(* IEC 61131-3 sources: teller/JD_Teller_LC2_V11/Class/TanabeCounterSerial, 1 file *)

(* ---- TanabeCounterSerial.st ---- *)
(*!
<Class
	Name               = "TanabeCounterSerial"
	Revision           = "1.0"
	RealtimeTask       = "false"
	CyclicTask         = "true"
	DefCyclictime      = "1 ms"
	BackgroundTask     = "false"
	Sigmatek           = "false"
	OSInterface        = "false"
	HighPriority       = "false"
	Automatic          = "false"
	UpdateMode         = "Prescan"
	SharedCommandTable = "true"
	Objectsize         = "(872,120)">
	<Channels>
		<Server Name="ClassSvr" Visualized="false" Initialize="false" WriteProtected="true" Retentive="false"/>
		<Server Name="iActualProduction" Visualized="false" Initialize="false" WriteProtected="false" Retentive="false"/>
		<Server Name="iBalanceOfProduction" Visualized="false" Initialize="false" WriteProtected="false" Retentive="false"/>
		<Server Name="iConveyorSpeed" Visualized="false" Initialize="false" WriteProtected="false" Retentive="false"/>
		<Server Name="iPlannedProduction" Visualized="false" Initialize="false" WriteProtected="false" Retentive="false"/>
		<Server Name="iProductionSpeed" Visualized="false" Initialize="false" WriteProtected="false" Retentive="false"/>
		<Server Name="sAangepasteWaarde" Visualized="false" Initialize="false" WriteProtected="false" Retentive="false"/>
		<Server Name="sBatch" Visualized="false" Initialize="false" WriteProtected="false" Retentive="false"/>
		<Server Name="sBattingDistance" Visualized="false" Initialize="false" WriteProtected="false" Retentive="false"/>
		<Server Name="sBattingStart" Visualized="false" Initialize="false" WriteProtected="false" Retentive="false"/>
		<Server Name="sBoxLength" Visualized="false" Initialize="false" WriteProtected="false" Retentive="false"/>
		<Server Name="sChangeOfActualQuantity" Visualized="false" Initialize="false" WriteProtected="true" Retentive="false"/>
		<Server Name="sCheckWrittenData" Visualized="false" Initialize="false" WriteProtected="true" Retentive="false"/>
		<Server Name="sClearProdData" Visualized="false" Initialize="false" WriteProtected="true" Retentive="false"/>
		<Server Name="sDateInput" Visualized="false" Initialize="false" WriteProtected="false" Retentive="false"/>
		<Server Name="sLotNo" Visualized="false" Initialize="false" WriteProtected="false" Retentive="false"/>
		<Server Name="sOperatorName" Visualized="false" Initialize="false" WriteProtected="false" Retentive="false"/>
		<Server Name="sProductionQuantity" Visualized="false" Initialize="false" WriteProtected="false" Retentive="false"/>
		<Server Name="sReadAConditionInProgress" Visualized="false" Initialize="false" WriteProtected="true" Retentive="false"/>
		<Server Name="sReturnNak" Visualized="false" Initialize="false" WriteProtected="true" Retentive="false"/>
		<Server Name="sStartingDistanceToConveyor" Visualized="false" Initialize="false" WriteProtected="false" Retentive="false"/>
		<Server Name="sTimeInput" Visualized="false" Initialize="false" WriteProtected="false" Retentive="false"/>
		<Server Name="sWriteProductionData" Visualized="false" Initialize="false" WriteProtected="true" Retentive="false"/>
		<Server Name="verklikker" Visualized="false" Initialize="false" WriteProtected="true" Retentive="false"/>
		<Server Name="Verzenden" Visualized="false" Initialize="false" WriteProtected="false" Retentive="false"/>
		<Client Name="cBatch1" Required="true" Internal="false"/>
		<Client Name="cBatch2" Required="true" Internal="false"/>
		<Client Name="cBattingDistance" Required="true" Internal="false"/>
		<Client Name="cBattingStart" Required="true" Internal="false"/>
		<Client Name="cBoxLength" Required="true" Internal="false"/>
		<Client Name="cCountedBoxes" Required="true" Internal="false"/>
		<Client Name="cPlannedProduction" Required="true" Internal="false"/>
		<Client Name="cStartingDistanceToConveyorRun" Required="true" Internal="false"/>
		<Client Name="FileBase" Required="true" Internal="false"/>
		<Client Name="GetInfo" Required="true" Internal="false"/>
		<Client Name="RxTx" Required="true" Internal="false"/>
		<Client Name="String" Required="true" Internal="false"/>
	</Channels>
	<RevDoku>
		<Owner Company="JD" Author="SV"/>
		<Dokumentation Revision="1" Date="2014-10-13" Author="SV" Company="JD" Description="Class om serieel (RS232) te communiceren met de hoofdcomputer van Tanabe."/>
	</RevDoku>
</Class>
*)
TanabeCounterSerial : CLASS
	TYPE
#pragma pack(push, 1)
	  TypeW : STRUCT  //! <Type Public="true" Name="TypeW"/>
	    Header : ARRAY [0..3] OF CHAR;
	    DateInput : ARRAY [0..6] OF CHAR;
	    TimeInPut : ARRAY [0..6] OF CHAR;
	    ProductionQuantity : ARRAY [0..6] OF CHAR;
	    BoxLength : ARRAY [0..4] OF CHAR;
	    BattingStart : ARRAY [0..3] OF CHAR;
	    BattingDistance : ARRAY [0..3] OF CHAR;
	    Batch : ARRAY [0..2] OF CHAR;
	    LotNo : ARRAY [0..17] OF CHAR;
	    OperatorName : ARRAY [0..8] OF CHAR;
	    StartingDistanceConveyor : ARRAY [0..4] OF CHAR;
	    AlterationOfActualProduction : ARRAY [0..6] OF CHAR;
	    Terminator : CHAR;
	  END_STRUCT;
#pragma pack(pop)
	END_TYPE
  //Servers:
	ClassSvr 	: SvrChCmd_DINT;
	verklikker 	: SvrCh_DINT;
	sReadAConditionInProgress 	: SvrCh_UDINT;
	sWriteProductionData 	: SvrCh_UDINT;
	sCheckWrittenData 	: SvrCh_UDINT;
	sClearProdData 	: SvrCh_UDINT;
	sChangeOfActualQuantity 	: SvrCh_UDINT;
	sReturnNak 	: SvrCh_UDINT;
	iPlannedProduction 	: SvrCh_DINT;
	iBalanceOfProduction 	: SvrCh_DINT;
	iActualProduction 	: SvrCh_DINT;
	iProductionSpeed 	: SvrCh_DINT;
	iConveyorSpeed 	: SvrCh_DINT;
	sDateInput 	: SvrCh_DINT;
	sTimeInput 	: SvrCh_DINT;
	sProductionQuantity 	: SvrCh_DINT;
	sBoxLength 	: SvrCh_DINT;
	sBattingStart 	: SvrCh_DINT;
	sBattingDistance 	: SvrCh_DINT;
	sBatch 	: SvrCh_DINT;
	sLotNo 	: SvrCh_DINT;
	sOperatorName 	: SvrCh_DINT;
	sStartingDistanceToConveyor 	: SvrCh_DINT;
	sAangepasteWaarde 	: SvrCh_DINT;
	Verzenden 	: SvrCh_DINT;
  //Clients:
	GetInfo 	: CltChCmd_TellerClass_Teller;
	RxTx 	: CltChCmd__SerLib;
	String 	: CltChCmd_String;
	FileBase 	: CltChCmd_FileBase;
	cPlannedProduction 	: CltCh_DINT;
	cBoxLength 	: CltCh_DINT;
	cBattingStart 	: CltCh_DINT;
	cBattingDistance 	: CltCh_DINT;
	cBatch1 	: CltCh_DINT;
	cBatch2 	: CltCh_DINT;
	cStartingDistanceToConveyorRun 	: CltCh_DINT;
	cCountedBoxes 	: CltCh_DINT;
  //Variables:
		ReadString1 : ARRAY [0..1] OF CHAR;

		ReadString2 : ARRAY [0..70] OF CHAR;

		SendStringToHost : ARRAY [0..70] OF CHAR;

		In1 : ARRAY [0..70] OF CHAR;

		VerifyData : ARRAY [0..4] OF CHAR;

		ConversieString : ARRAY [0..20] OF CHAR;

		VulString : ARRAY [0..20] OF CHAR;

		ReadAConditionInProgress : ARRAY [0..4] OF CHAR;
			//! <Variable Comment="Read a condition in progress." Name="ReadAConditionInProgress"/>
		ReturnReadAConditionInProgress : ARRAY [0..35] OF CHAR;

		WriteProductionData 	: TypeW;
		ClearProdData : ARRAY [0..4] OF CHAR;

		ChangeOfActualProducedQuantity : ARRAY [0..4] OF CHAR;

		S_ : ARRAY [0..4] OF CHAR;

		ReturnS_ : ARRAY [0..4] OF CHAR;

		rdlenVar 	: UDINT;
		receivedLen 	: UDINT;
		ReadIndex 	: UDINT;
		ClearIndex 	: DINT;
		Index 	: UDINT;
		index2 	: UDINT;
		Poll 	: CHAR;
		TimeMark 	: UDINT;
		Delaytime 	: UDINT;
		Stringlengte 	: UDINT;
		udByteSend 	: UDINT;
		KnopOud 	: DINT;
		In2 	: DINT;
		In3 	: DINT;
		InIndex 	: DINT;
		S_2 : ARRAY [0..3] OF CHAR;

		Timemark2 	: UDINT;
		DelayTime2 	: UDINT;
  //Functions:

	FUNCTION VIRTUAL GLOBAL Init;

	FUNCTION VIRTUAL GLOBAL CyWork
		VAR_INPUT
			EAX 	: UDINT;
		END_VAR
		VAR_OUTPUT
			state (EAX) 	: UDINT;
		END_VAR;

	FUNCTION ClrReadString1_2;

	FUNCTION ClrSendStringToHost;

	FUNCTION ClrConversie_Vulstring;

	FUNCTION ClrIn1;

	FUNCTION WriteDataToCounter;
  //Tables:
	FUNCTION @STD
		VAR_OUTPUT
			ret_code	: CONFSTATES;
		END_VAR;
	FUNCTION GLOBAL TAB @CT_;
END_CLASS;

#pragma usingLtd _SerLib
#pragma usingLtd FileBase
#pragma usingLtd String
#pragma usingLtd TellerClass_Teller

FUNCTION VIRTUAL GLOBAL TanabeCounterSerial::Init
VAR
	i : UDINT;

END_VAR

if _FirstScan then

RxTx.StartUser(Baud:= SERUSERBAUD_9600, wordl:= 8, Parity:= SERUSERPARITY_NONE, StopB:= 1, FifoOnOff:= 0);
RxTx.SetRSMode(Mode:=232);

//Header data van teller opvragen
ReadAConditionInProgress[0] := 2;
ReadAConditionInProgress[1] := 'D';
ReadAConditionInProgress[2] := 'C';
ReadAConditionInProgress[3] := 'R';
ReadAConditionInProgress[4] := 13;

//Header data vanaf hoofdcomputer
WriteProductionData.Header[0] := 2;
WriteProductionData.Header[1] := 'D';
WriteProductionData.Header[2] := 'C';
WriteProductionData.Header[3] := 'W';
WriteProductionData.Terminator:= 13;

//Header aanvraag voor verificatie
VerifyData[0] := 2;
VerifyData[1] := 'D';
VerifyData[2] := 'C';
VerifyData[3] := 'V';
VerifyData[4] := 13;

//Data nullen commando
ClearProdData[0] := 2;
ClearProdData[1] := 'D';
ClearProdData[2] := 'C';
ClearProdData[3] := 'C';
ClearProdData[4] := 13;

//Header change of actul produced quantity
ChangeOfActualProducedQuantity[0] := 2;
ChangeOfActualProducedQuantity[1] := 'D';
ChangeOfActualProducedQuantity[2] := 'C';
ChangeOfActualProducedQuantity[3] := 'A';
ChangeOfActualProducedQuantity[4] := 13;

//Vraag voor NAK
S_[0] := 2;
S_[1] := 'D';
S_[2] := 'C';
S_[3] := 'S';
S_[4] := 13;

S_2[0] := 2;
S_2[1] := 'D';
S_2[2] := 'C';
S_2[3] := 13;
//S_[4] := 13;

//Antwoord op S_(NAK, ascii 21).
ReturnS_[0] := 2;
ReturnS_[1] := 'D';
ReturnS_[2] := 'C';
ReturnS_[3] := 21;
ReturnS_[4] := 13;

for i := 0 to 20 do
 VulString[i] := '0';
end_for;

Delaytime := 500; //verklikker
TimeMark := 0;
Delaytime2 := 150;
TimeMark2 := 0;
end_if;

END_FUNCTION

FUNCTION VIRTUAL GLOBAL TanabeCounterSerial::CyWork
	VAR_INPUT
		EAX 	: UDINT;
	END_VAR
	VAR_OUTPUT
		state (EAX) 	: UDINT;
	END_VAR

//waarden uit de tellerClass_teller halen die nodig zijn voor DCR
iPlannedProduction := GetInfo.sTotalProduction;
iBalanceOfProduction := GetInfo.sRemainingProduction;
iActualProduction := GetInfo.sCounter;
iProductionSpeed := GetInfo.sCounterPerMin;
iConveyorSpeed := 1;//

//kijken of er data beschikbaar is.
receivedLen := RxTx.GetRecvState();

//als er data is dan:
if receivedLen > 0 then
  //data naar buffer
  RxTx.RecvBlock(Buffer:=#ReadString1[0], rdlength:= receivedLen, rdlen:=#rdlenVar);
  //copieer data naar string
  _memcpy(ptr1:=#ReadString2[ReadIndex], ptr2:=#ReadString1[0], cntr:=receivedLen);

  //ReadIndex ophogen
  ReadIndex += receivedLen ;

end_if;

//RETURN READ A CONDITION IN PROGRESS
sReadAConditionInProgress := _memcmp(ptr1:=#ReadString2, ptr2:=#ReadAConditionInProgress, cntr:= _strlen(src:=#ReadAConditionInProgress[0]));

if sReadAConditionInProgress = 0 then

if ops.tAbsolute - Timemark2 > DelayTime2 then
Timemark2 := ops.tAbsolute;
ClrSendStringToHost();

SendStringToHost[0] := 2;
SendStringToHost[1] := 'D';
SendStringToHost[2] := 'C';

FileBase.BuildValue2Ascii(Value:=iPlannedProduction, Dest:=#ConversieString[0], Offset:=0);
_memcpy(ptr1:=#VulString[_strlen(src:=#VulString[0]) - _strlen(src:=#ConversieString[0])], ptr2:=#ConversieString[0], cntr:= _strlen(src:=#ConversieString[0]));
_memcpy(ptr1:=#SendStringToHost[3], ptr2:=#VulString[15], cntr:=6);
ClrConversie_Vulstring();

FileBase.BuildValue2Ascii(Value:=iBalanceOfProduction, Dest:=#ConversieString[0], Offset:=0);
_memcpy(ptr1:=#VulString[_strlen(src:=#VulString[0]) - _strlen(src:=#ConversieString[0])], ptr2:=#ConversieString[0], cntr:= _strlen(src:=#ConversieString[0]));
_memcpy(ptr1:=#SendStringToHost[9], ptr2:=#VulString[15], cntr:=6);
ClrConversie_Vulstring();

FileBase.BuildValue2Ascii(Value:=iActualProduction, Dest:=#ConversieString[0], Offset:=0);
_memcpy(ptr1:=#VulString[_strlen(src:=#VulString[0]) - _strlen(src:=#ConversieString[0])], ptr2:=#ConversieString[0], cntr:= _strlen(src:=#ConversieString[0]));
_memcpy(ptr1:=#SendStringToHost[15], ptr2:=#VulString[15], cntr:=6);
ClrConversie_Vulstring();

FileBase.BuildValue2Ascii(Value:=iProductionSpeed, Dest:=#ConversieString[0], Offset:=0);
_memcpy(ptr1:=#VulString[_strlen(src:=#VulString[0]) - _strlen(src:=#ConversieString[0])], ptr2:=#ConversieString[0], cntr:= _strlen(src:=#ConversieString[0]));
_memcpy(ptr1:=#SendStringToHost[21], ptr2:=#VulString[15], cntr:=6);
ClrConversie_Vulstring();

FileBase.BuildValue2Ascii(Value:=iConveyorSpeed, Dest:=#ConversieString[0], Offset:=0);
_memcpy(ptr1:=#VulString[_strlen(src:=#VulString[0]) - _strlen(src:=#ConversieString[0])], ptr2:=#ConversieString[0], cntr:= _strlen(src:=#ConversieString[0]));
_memcpy(ptr1:=#SendStringToHost[27], ptr2:=#VulString[15], cntr:=6);
ClrConversie_Vulstring();

SendStringToHost[33] := 13;
Verzenden := 1;

end_if;
end_if;

//WRITE DATA VANAF TANABE
sWriteProductionData := _memcmp(ptr1:=#ReadString2[0], ptr2:=#WriteProductionData.Header, cntr:= 4 );
if sWriteProductionData = 0 then

//sProductionQuantity := 0;
//sBoxLength := 0;
//sBattingStart := 0;
//sBattingDistance := 0;
//sBatch:= 0;
//sLotNo := 0;
//sOperatorName := 0;
//sStartingDistanceToConveyor:= 0;
//sAangepasteWaarde := 0;

_memcpy(ptr1:=#WriteProductionData.DateInput[0], ptr2:=#ReadString2[4], cntr:=6);_memcpy(ptr1:=#WriteProductionData.TimeInPut[0], ptr2:=#ReadString2[10], cntr:=6);
_memcpy(ptr1:=#WriteProductionData.ProductionQuantity[0], ptr2:=#ReadString2[16], cntr:=6);
_memcpy(ptr1:=#WriteProductionData.BoxLength[0], ptr2:=#ReadString2[22], cntr:=4);
_memcpy(ptr1:=#WriteProductionData.BattingStart[0], ptr2:=#ReadString2[26], cntr:=3);
_memcpy(ptr1:=#WriteProductionData.BattingDistance[0], ptr2:=#ReadString2[29], cntr:=3);
_memcpy(ptr1:=#WriteProductionData.Batch[0], ptr2:=#ReadString2[32], cntr:=2);
_memcpy(ptr1:=#WriteProductionData.LotNo[0], ptr2:=#ReadString2[34], cntr:=17);
_memcpy(ptr1:=#WriteProductionData.OperatorName[0], ptr2:=#ReadString2[51], cntr:=8);
_memcpy(ptr1:=#WriteProductionData.StartingDistanceConveyor[0], ptr2:=#ReadString2[59], cntr:=4);

sDateInput :=  filebase.ConvAscii2Value(Source:=#WriteProductionData.DateInput[0]);
sTimeInput :=  filebase.ConvAscii2Value(Source:=#WriteProductionData.TimeInPut[0]);
sProductionQuantity :=  filebase.ConvAscii2Value(Source:=#WriteProductionData.ProductionQuantity[0]);
sBoxLength :=  filebase.ConvAscii2Value(Source:=#WriteProductionData.BoxLength[0]);
sBattingStart := FileBase.ConvAscii2Value(Source:=#WriteProductionData.BattingStart[0]);
sBattingDistance :=  filebase.ConvAscii2Value(Source:=#WriteProductionData.BattingDistance[0]);
sBatch := FileBase.ConvAscii2Value(Source:=#WriteProductionData.Batch[0]);
sLotNo := filebase.ConvAscii2Value(Source:=#WriteProductionData.LotNo[0]);
sOperatorName :=  filebase.ConvAscii2Value(Source:=#WriteProductionData.OperatorName[0]);
sStartingDistanceToConveyor :=  filebase.ConvAscii2Value(Source:=#WriteProductionData.StartingDistanceConveyor[0]);

cPlannedProduction := sProductionQuantity;
cBoxLength := sBoxLength;
cBattingStart := sBattingStart;
cBattingDistance := sBattingDistance;
cBatch1 := sBatch;
cBatch2 := 0;
cStartingDistanceToConveyorRun := sStartingDistanceToConveyor;
cCountedBoxes := 0;

WriteDataToCounter();

end_if;

//VERIFY WRITTEN DATA
sCheckWrittenData := _memcmp(ptr1:=#ReadString2, ptr2:=#VerifyData[0], cntr:=4);
if sCheckWrittenData = 0 then

ClrSendStringToHost();

//ClrOperatorLorNo();

SendStringToHost[0] := 2;
SendStringToHost[1] := 'D';
SendStringToHost[2] := 'C';

FileBase.BuildValue2Ascii(Value:=sDateInput, Dest:=#ConversieString[0], Offset:=0);
_memcpy(ptr1:=#VulString[_strlen(src:=#VulString[0]) - _strlen(src:=#ConversieString[0])], ptr2:=#ConversieString[0], cntr:= _strlen(src:=#ConversieString[0]));
_memcpy(ptr1:=#SendStringToHost[3], ptr2:=#VulString[15], cntr:=6);
ClrConversie_Vulstring();

FileBase.BuildValue2Ascii(Value:=sTimeInput, Dest:=#ConversieString[0], Offset:=0);
_memcpy(ptr1:=#VulString[_strlen(src:=#VulString[0]) - _strlen(src:=#ConversieString[0])], ptr2:=#ConversieString[0], cntr:= _strlen(src:=#ConversieString[0]));
_memcpy(ptr1:=#SendStringToHost[9], ptr2:=#VulString[15], cntr:=6);
ClrConversie_Vulstring();

FileBase.BuildValue2Ascii(Value:=sProductionQuantity, Dest:=#ConversieString[0], Offset:=0);
_memcpy(ptr1:=#VulString[_strlen(src:=#VulString[0]) - _strlen(src:=#ConversieString[0])], ptr2:=#ConversieString[0], cntr:= _strlen(src:=#ConversieString[0]));
_memcpy(ptr1:=#SendStringToHost[15], ptr2:=#VulString[15], cntr:=6);
ClrConversie_Vulstring();

FileBase.BuildValue2Ascii(Value:=sBoxLength, Dest:=#ConversieString[0], Offset:=0);
_memcpy(ptr1:=#VulString[_strlen(src:=#VulString[0]) - _strlen(src:=#ConversieString[0])], ptr2:=#ConversieString[0], cntr:= _strlen(src:=#ConversieString[0]));
_memcpy(ptr1:=#SendStringToHost[21], ptr2:=#VulString[17], cntr:=4);
ClrConversie_Vulstring();

//FileBase.BuildValue2Ascii(Value:=sBattingStart, Dest:=#ConversieString[0], Offset:=0);
//_memcpy(ptr1:=#VulString[_strlen(src:=#VulString[0]) - _strlen(src:=#ConversieString[0])], ptr2:=#ConversieString[0], cntr:= _strlen(src:=#ConversieString[0]));
//_memcpy(ptr1:=#SendStringToHost[25], ptr2:=#VulString[18], cntr:=3);
//ClrConversie_Vulstring();

FileBase.BuildValue2Ascii(Value:=sBattingDistance, Dest:=#ConversieString[0], Offset:=0);
_memcpy(ptr1:=#VulString[_strlen(src:=#VulString[0]) - _strlen(src:=#ConversieString[0])], ptr2:=#ConversieString[0], cntr:= _strlen(src:=#ConversieString[0]));
_memcpy(ptr1:=#SendStringToHost[25], ptr2:=#VulString[19], cntr:=2);
ClrConversie_Vulstring();

//FileBase.BuildValue2Ascii(Value:=sBatch, Dest:=#ConversieString[0], Offset:=0);
//_memcpy(ptr1:=#VulString[_strlen(src:=#VulString[0]) - _strlen(src:=#ConversieString[0])], ptr2:=#ConversieString[0], cntr:= _strlen(src:=#ConversieString[0]));
//_memcpy(ptr1:=#SendStringToHost[31], ptr2:=#VulString[19], cntr:=2);
//ClrConversie_Vulstring();

FileBase.BuildValue2Ascii(Value:=sLotNo, Dest:=#ConversieString[0], Offset:=0);
_memcpy(ptr1:=#VulString[_strlen(src:=#VulString[0]) - _strlen(src:=#ConversieString[0])], ptr2:=#ConversieString[0], cntr:= _strlen(src:=#ConversieString[0]));
_memcpy(ptr1:=#SendStringToHost[27], ptr2:=#VulString[4], cntr:=17);
ClrConversie_Vulstring();

FileBase.BuildValue2Ascii(Value:=sOperatorName, Dest:=#ConversieString[0], Offset:=0);
_memcpy(ptr1:=#VulString[_strlen(src:=#VulString[0]) - _strlen(src:=#ConversieString[0])], ptr2:=#ConversieString[0], cntr:= _strlen(src:=#ConversieString[0]));
_memcpy(ptr1:=#SendStringToHost[44], ptr2:=#VulString[13], cntr:=8);
ClrConversie_Vulstring();

FileBase.BuildValue2Ascii(Value:=sStartingDistanceToConveyor, Dest:=#ConversieString[0], Offset:=0);
_memcpy(ptr1:=#VulString[_strlen(src:=#VulString[0]) - _strlen(src:=#ConversieString[0])], ptr2:=#ConversieString[0], cntr:= _strlen(src:=#ConversieString[0]));
_memcpy(ptr1:=#SendStringToHost[52], ptr2:=#VulString[17], cntr:=4);
ClrConversie_Vulstring();

//  CHANGE OF ACTUAL VALUE???????
FileBase.BuildValue2Ascii(Value:=sAangepasteWaarde, Dest:=#ConversieString[0], Offset:=0);
_memcpy(ptr1:=#VulString[_strlen(src:=#VulString[0]) - _strlen(src:=#ConversieString[0])], ptr2:=#ConversieString[0], cntr:= _strlen(src:=#ConversieString[0]));
_memcpy(ptr1:=#SendStringToHost[56], ptr2:=#VulString[15], cntr:=6);
ClrConversie_Vulstring();

SendStringToHost[62] := 13;
Verzenden := 1;
end_if;

//CLEAR DATA (DCC)
sClearProdData := _memcmp(ptr1:=#ReadString2, ptr2:=#ClearProdData[0], cntr:= 4 );
if sClearProdData = 0 then

  sProductionQuantity := 0;
  sBoxLength := 0;
  sBattingStart := 0;
  sBattingDistance := 0;
  sBatch:= 0;
  sLotNo := 0;
  sOperatorName := 0;
  sStartingDistanceToConveyor:= 0;
  sAangepasteWaarde := 0;

cPlannedProduction := sProductionQuantity;
cBoxLength := sBoxLength;
cBattingStart := sBattingStart;
cBattingDistance := sBattingDistance;
cBatch1 := sBatch;
cBatch2 := 0;
cStartingDistanceToConveyorRun := sStartingDistanceToConveyor;
cCountedBoxes := 0;

WriteDataToCounter();

end_if;

//CHANGE OF ACTUAL PRODUCED QUANTITY (DCA)
sChangeOfActualQuantity := _memcmp(ptr1:=#ReadString2[0], ptr2:=#ChangeOfActualProducedQuantity, cntr:= 4 );
if sChangeOfActualQuantity = 0 then
  _memcpy(ptr1:=#WriteProductionData.AlterationOfActualProduction[0], ptr2:=#ReadString2[4], cntr:=6);
  sAangepasteWaarde :=  filebase.ConvAscii2Value(Source:=#WriteProductionData.AlterationOfActualProduction[0]);
end_if;

//RETURN A NEGATIVE ACKNOWLEDGEMENT (NAK)
sReturnNak := _memcmp(ptr1:=#ReadString2[0], ptr2:=#S_, cntr:= _strlen(src:=#S_[0]))| _memcmp(ptr1:=#ReadString2[0], ptr2:=#S_2, cntr:= 3);
if sReturnNak = 0 then
  ClrSendStringToHost();
  _memcpy(ptr1:=#SendStringToHost[0], ptr2:=#ReturnS_[0], cntr:= 5);
  Verzenden := 1;
  // RxTx.SerSend(Buffer:=#SendStringToHost[0], Bufferlength:= _strlen(src:=#ReturnS_[0]), WrLen:=#udByteSend);
end_if;

//kijken of er een 13 (CR) is
Poll := ReadString2[Index];
Index += 1;
  if index >=  _strlen(src:=#ReadString2[0]) then
   Index := 0;
 end_if;

//zo ja, stringen leegmaken.
if Poll = 13 then
ClrIn1();
_memcpy(ptr1:=#In1[0], ptr2:=#ReadString2, cntr:=70);
ClrReadString1_2();
end_if;

//verklikker of er een commando string binnenkomt.
if sReadAConditionInProgress = 0 |
        sWriteProductionData = 0 |
              sClearProdData = 0 |
                  sReturnNak = 0 |
     sChangeOfActualQuantity = 0 |
           sCheckWrittenData = 0

then
  verklikker := 1;
  TimeMark := ops.tAbsolute;
end_if;

if ops.tAbsolute - TimeMark > Delaytime then
  verklikker := 0;
end_if;

if Verzenden = 1 then
  RxTx.SerSend(Buffer:=#SendStringToHost[0], Bufferlength:=_strlen(src:=#SendStringToHost[0]), WrLen:=#udByteSend);
  Verzenden := 0;
end_if;

state := READY;

END_FUNCTION

FUNCTION TanabeCounterSerial::ClrReadString1_2

VAR
	i : UDINT;
  ii : int;
END_VAR

for i := 0 to 65 do
  ReadString2[i] := 0;
end_for;

for ii := 0 to 1 do
  ReadString1[ii] := 0;
end_for;

ReadIndex := 0;

END_FUNCTION

FUNCTION TanabeCounterSerial::ClrSendStringToHost

VAR
	i : int;
END_VAR

for i := 0 to 70 do
  SendStringToHost[i] := 0;
end_for;

END_FUNCTION

FUNCTION TanabeCounterSerial::ClrConversie_Vulstring
VAR
	i : int;
END_VAR

for i := 0 to 20 do
  ConversieString[i] := 0;
  VulString[i]       := '0';
end_for;

END_FUNCTION

FUNCTION TanabeCounterSerial::ClrIn1
VAR
	i : int;
END_VAR

for i := 0 to 65 do
  In1[i] := 0;

end_for;

END_FUNCTION

FUNCTION TanabeCounterSerial::WriteDataToCounter

cPlannedProduction.Write (cPlannedProduction);
cBoxLength.Write (cBoxLength);
cBattingStart.Write (cBattingStart);
cBattingDistance.Write (cBattingDistance);
cBatch1.Write (cBatch1);
cBatch2.Write (cBatch2);
cStartingDistanceToConveyorRun.Write (cStartingDistanceToConveyorRun);
cCountedBoxes.Write (cCountedBoxes);

END_FUNCTION
